// TIA Portal V20 export
VAR_GLOBAL   // PLC tag table "Unit1Em6"
   "BA010AZCRPM04.12" AT %Q2013.2 : Bool;   // VISION PUSHER SUPPORT DOWN
   "BA010AZCRPM04.13" AT %Q2013.3 : Bool;   // VISION PUSHER SUPPORT UP
   "BA010AZCRBK05.05" AT %I1016.5 : Bool;   // VISION PUSHER SUPPORT UP
   "BA010AZCRBK05.15" AT %I1017.5 : Bool;   // VISION PUSHER SUPPORT DOWN
   "BA010AZCRSP506.02" AT %I3300.2 : Bool;   // VISION TRIGGER SENSOR
   "BA010AZCRSP501.04" AT %I3000.4 : Bool;   // Vision STO // STO - 판정 결과때 같이 살음
   "BA010AZCRSP501.05" AT %I3000.5 : Bool;   // VISION JUDGMENT // TRUE = NG, FALSE= OK
   "BA010AZCRSP506.06" AT %Q3300.2 : Bool;   // VISION CONTROLLER TRIGGER
END_VAR
VAR_GLOBAL CONSTANT   // user constants
   U1EM6_NO_OF_AXES : USInt := 1;   // Starts with 1. E.g., the value 4 means that 4 axes exist.
   DR9_RatedTorque : LReal := 1.27;   // VisionAxisZ
   U1EM6_JOB01 : DInt := 1;
   U1EM6_JOB02 : DInt := 2;
   U1EM6_JOB03 : DInt := 3;
   U1EM6_JOB04 : DInt := 4;
   U1EM6_JOB05 : DInt := 5;
   U1EM6_JOB06 : DInt := 6;
   U1EM6_JOB07 : DInt := 7;
   U1EM6_JOB08 : DInt := 8;
   U1EM6_JOB09 : DInt := 9;
   U1EM6_JOB10 : DInt := 10;
   U1EM6_JOB11 : DInt := 11;
   U1EM6_JOB12 : DInt := 12;
   U1EM6_JOB13 : DInt := 13;
   U1EM6_JOB14 : DInt := 14;
   U1EM6_JOB15 : DInt := 15;
   U1EM6_JOB16 : DInt := 16;
   U1EM6_JOB17 : DInt := 17;
   U1EM6_JOB18 : DInt := 18;
   U1EM6_JOB19 : DInt := 19;
   U1EM6_JOB20 : DInt := 20;
   U1EM6_JOB21 : DInt := 21;
   U1EM6_JOB22 : DInt := 22;
   U1EM6_JOB23 : DInt := 23;
   U1EM6_JOB24 : DInt := 24;
   U1EM6_JOB25 : DInt := 25;
   U1EM6_JOB26 : DInt := 26;
   U1EM6_JOB27 : DInt := 27;
   U1EM6_JOB28 : DInt := 28;
   U1EM6_JOB29 : DInt := 29;
   U1EM6_JOB30 : DInt := 30;
   U1EM6_JOB31 : DInt := 31;
   U1EM6_JOB32 : DInt := 32;
   U1EM6_JOB33 : DInt := 33;
   U1EM6_JOB34 : DInt := 34;
   U1EM6_JOB35 : DInt := 35;
   U1EM6_JOB36 : DInt := 36;
   U1EM6_JOB37 : DInt := 37;
   U1EM6_JOB38 : DInt := 38;
   U1EM6_JOB39 : DInt := 39;
   U1EM6_JOB40 : DInt := 40;
   U1EM6_JOB41 : DInt := 41;
   U1EM6_JOB42 : DInt := 42;
   U1EM6_JOB43 : DInt := 43;
   U1EM6_JOB44 : DInt := 44;
   U1EM6_JOB45 : DInt := 45;
   U1EM6_JOB46 : DInt := 46;
   U1EM6_JOB47 : DInt := 47;
   U1EM6_JOB48 : DInt := 48;
   U1EM6_JOB49 : DInt := 49;
   U1EM6_JOB50 : DInt := 50;
END_VAR
